{attribute addProperty BoxType "EL6851-0010-0016"}
{attribute addProperty Id "ChannelAT %I*ARRAY[0 ..63] OF USINT512640"}
{attribute addProperty CRC "2702512740"}
{attribute addProperty SizeInBites "512"}
{attribute addProperty SizeInBytes "64"}
TYPE DMX_Channel_D03720FB :
STRUCT
	{attribute addProperty Name "Channel"}
	Channel AT %I* : ARRAY[0 ..63] OF USINT;
END_STRUCT
END_TYPE

(* stored: Version 1.2.0.0, ProductVersion 3.1.4024.9
   DUT DMX_Channel_D03720FB: Id {aab9c82a-0c67-4a2b-a47d-6a02ff73f5e6} *)
